Fanuc KAREL source: VAR_INFO.kl

PROGRAM T
%NOLOCKGROUP
VAR
 v0 : STRING[40]
 v1 : STRING[40]
 v2 : BOOLEAN
 v3 : STRING[40]
 v4 : INTEGER
 v5 : ARRAY[3] OF INTEGER
 v6 : INTEGER
 v7 : INTEGER
BEGIN
 VAR_INFO(v0, v1, v2, v3, v4, v5, v6, v7)
END T
